FUNCTION_BLOCK MC_SmoothMover
VAR_IN_OUT
    Axis	:	AXIS_REF;
END_VAR
VAR_INPUT
    Velocity : LREAL;
    ReqAbsPos : LREAL; //A
    Enable	:	BOOL; //While true the block will accept new positions and attempt to move to them if they are different
    Execute	:	BOOL; //Will retry a move if the target position is the same
END_VAR
VAR_OUTPUT
    Done	:	BOOL;
    Busy	:	BOOL;
    Error	:	BOOL;
END_VAR
VAR
    mcMoveAbsolute : ARRAY[1..2] OF MC_MoveAbsolute;
    iI: INT;
    imcBlockIndex: INT;
    ReqAbsPosPrevious	: LREAL;
    rtExecute: R_TRIG;
END_VAR

(* Smooth Mover
2017-8-30
A. Wallace

Enable means the block will always aquire new positions as they are updated. Execute
can be used to retry a move.
*)


rtExecute(CLK:=Execute);

IF ( (ReqAbsPos <> ReqAbsPosPrevious AND Enable) OR rtExecute.Q) THEN
            mcMoveAbsolute[imcBlockIndex].Execute := FALSE;
            imcBlockIndex := imcBlockIndex + 1;
            IF imcBlockIndex >2 THEN imcBlockIndex := 1; END_IF
            mcMoveAbsolute[imcBlockIndex].Position := ReqAbsPos;
            mcMoveAbsolute[imcBlockIndex].Execute := TRUE;
            ReqAbsPosPrevious := ReqAbsPos;
        ELSIF mcMoveAbsolute[imcBlockIndex].Done OR
                mcMoveAbsolute[imcBlockIndex].CommandAborted OR
                mcMoveAbsolute[imcBlockIndex].Busy OR
                mcMoveAbsolute[imcBlockIndex].Error THEN
            mcMoveAbsolute[imcBlockIndex].Execute := FALSE;
        END_IF

FOR iI := 1 TO 2 DO
    mcMoveAbsolute[iI](Axis := Axis, Velocity:=Velocity, BufferMode:=MC_Aborting);
END_FOR

Error := mcMoveAbsolute[1].Error OR mcMoveAbsolute[2].Error;
Done S= mcMoveAbsolute[1].Done OR mcMoveAbsolute[2].Done;
Busy := mcMoveAbsolute[1].Busy OR mcMoveAbsolute[2].Busy;
Done R= Busy OR Error;

END_FUNCTION_BLOCK

(* stored: Version 1.1.0.1, ProductVersion 3.1.4020.12
   POU MC_SmoothMover: Id {49439872-0161-4fd4-9e7f-62bcb9508941}, SpecialFunc None *)
